PROGRAM Stn053_PrgCalls
VAR
END_VAR

//Turn on the default programs
IF gFirstScan THEN
	gDebug_ComponentCalls.CallStn053_22_EvalBreakStopsBlu := TRUE;
	gDebug_ComponentCalls.CallStn053_25_EmptyPuckStorageBreakStop1Red := TRUE;
	gDebug_ComponentCalls.CallStn053_26_EmptyPuckStorageBreakStop2Red := TRUE;
	gDebug_ComponentCalls.CallStn053_41_BufferRecircMainMergePrestopRed := TRUE;
	gDebug_ComponentCalls.CallStn053_42_BufferRecircSpurMergePrestopRed := TRUE;
	gDebug_ComponentCalls.CallStn053_43_BufferRecircMergeRed := TRUE;
	gDebug_ComponentCalls.CallStn053_45_CleaningRecircExitDivertRed := TRUE;
	gDebug_ComponentCalls.CallStn053_98_ReceivingBypassExitMergeMainPrestopBlu := TRUE;
	gDebug_ComponentCalls.CallStn053_99_ReceivingBypassExitMergeBlu := TRUE;
END_IF

// Call Components
IF gDebug_ComponentCalls.CallStn053_22_EvalBreakStopsBlu OR
		gFirstScan THEN
	Stn053_22_EvalBreakStopsBlu();
END_IF
IF gDebug_ComponentCalls.CallStn053_25_EmptyPuckStorageBreakStop1Red OR
		gFirstScan THEN
	Stn053_25_EmptyPuckStorageBreakStop1Red();
END_IF
IF gDebug_ComponentCalls.CallStn053_26_EmptyPuckStorageBreakStop2Red OR
		gFirstScan THEN
	Stn053_26_EmptyPuckStorageBreakStop2Red();
END_IF

IF gDebug_ComponentCalls.CallStn053_41_BufferRecircMainMergePrestopRed OR
		gFirstScan THEN
	Stn053_41_BufferRecircMainMergePrestopRed();
END_IF
IF gDebug_ComponentCalls.CallStn053_42_BufferRecircSpurMergePrestopRed OR
		gFirstScan THEN
	Stn053_42_BufferRecircSpurMergePrestopRed();
END_IF
IF gDebug_ComponentCalls.CallStn053_43_BufferRecircMergeRed OR
		gFirstScan THEN
	Stn053_43_BufferRecircMergeRed();
END_IF
IF gDebug_ComponentCalls.CallStn053_45_CleaningRecircExitDivertRed OR
		gFirstScan THEN
	Stn053_45_CleaningRecircExitDivertRed();
END_IF
IF gDebug_ComponentCalls.CallStn053_98_ReceivingBypassExitMergeMainPrestopBlu OR
		gFirstScan THEN
	Stn053_98_ReceivingBypassExitMergeMainPrestopBlu();
END_IF
IF gDebug_ComponentCalls.CallStn053_99_ReceivingBypassExitMergeBlu OR
		gFirstScan THEN
	Stn053_99_ReceivingBypassExitMergeBlu();
END_IF

END_PROGRAM

(* stored: Version 1.1.0.1, ProductVersion 3.1.4024.6
   POU Stn053_PrgCalls: Id {fc97e9f3-6060-42cf-b0d4-ed831a4455c7}, SpecialFunc None *)
